// TIA Portal project "Vagoneta-1516" (V15.1)

(* hardware
DEVICE "S71500/ET200MP station_1"  S7-1500 station
   slot 0: "Perfil soporte_0"  Rack  6ES7 590-1***0-0AA0
   slot 1: "PLC_1"  CPU 1516-3 PN/DP  6ES7 516-3AN01-0AB0  V2.6
      slot 3: "Display de la CPU_1"  6ES7591-1BA00-0AA0
*)

// ===== PLC "PLC_1"  CPU 1516-3 PN/DP =====

VAR_GLOBAL   // PLC tag table "Tabla de variables estándar"
   "E0-Reposo" AT %M10.0 : Bool;
   "E1-avance_a_carga" AT %M10.1 : Bool;
   "E2-carga" AT %M10.2 : Bool;
   "E3-avance_a_descarga" AT %M10.3 : Bool;
   "E4-descarga" AT %M10.4 : Bool;
   "P_marcha" AT %I0.0 : Bool;
   "FC1_inicio" AT %I0.1 : Bool;
   "FC2_carga" AT %I0.2 : Bool;
   "FC3_descarga" AT %I0.3 : Bool;
   "Luz_verde" AT %Q0.0 : Bool;
   "Luz_roja" AT %Q0.1 : Bool;
   "Valvula" AT %Q0.2 : Bool;
   "E5-retroceso" AT %M10.5 : Bool;
   "Tag_1" AT %M50.0 : Bool;
   "Tag_2" AT %M50.1 : Bool;
   "Tag_3" AT %M50.2 : Bool;
   "P_Paro" AT %I0.4 : Bool;
   "Motor_avanza" AT %Q0.3 : Bool;
   "Motor_retrocede" AT %Q0.4 : Bool;
   "Zumbador" AT %Q0.5 : Bool;
   "Error_www" AT %MW100 : Int;
   "ContadorCiclos" AT %MB102 : SInt;
   "Tag_4" AT %M50.6 : Bool;
   "Tag_5" AT %M50.3 : Bool;
   "Estado" AT %MB103 : SInt;
   "Tag_6" AT %M70.0 : Bool;
   "Tag_7" AT %M70.1 : Bool;
   "Tag_8" AT %M70.2 : Bool;
   "Tag_9" AT %M70.3 : Bool;
   "Tag_10" AT %M70.4 : Bool;
   "Tag_11" AT %M70.5 : Bool;
   "System_Byte" AT %MB1 : Byte;
   "FirstScan" AT %M1.0 : Bool;
   "DiagStatusUpdate" AT %M1.1 : Bool;
   "AlwaysTRUE" AT %M1.2 : Bool;
   "AlwaysFALSE" AT %M1.3 : Bool;
   "tCarga" AT %MW104 : Int;
   "tDescarga" AT %MW106 : Int;
END_VAR

// folder: System blocks/Program resources

DATA_BLOCK "TP_5s"   // DB1
{ S7_Optimized_Access := 'TRUE' }
AUTHOR : Simatic
FAMILY : IEC
NAME : IEC_TMR
VERSION : 1.0
// stored: InstanceOfName IEC_TIMER
"IEC_TIMER"
BEGIN
END_DATA_BLOCK

DATA_BLOCK "TP_descarga"   // DB2
{ S7_Optimized_Access := 'TRUE' }
AUTHOR : Simatic
FAMILY : IEC
NAME : IEC_TMR
VERSION : 1.0
// stored: InstanceOfName IEC_TIMER
"IEC_TIMER"
BEGIN
END_DATA_BLOCK

DATA_BLOCK "CTU_ciclos"   // DB3
{ S7_Optimized_Access := 'TRUE' }
AUTHOR : Simatic
FAMILY : IEC
NAME : CNTR
VERSION : 1.0
// stored: InstanceOfName IEC_COUNTER
"IEC_COUNTER"
BEGIN
END_DATA_BLOCK

// folder: (top level)

ORGANIZATION_BLOCK "Main"   // OB1, LAD, ProgramCycle
TITLE = "Main Program Sweep (Cycle)"
{ S7_Optimized_Access := 'TRUE' }
VERSION : 0.1
   VAR_INPUT
      Initial_Call : Bool;   // Initial call of this OB
      Remanence : Bool;   // =True, if remanent data are available
   END_VAR
   VAR_TEMP   // added for the SCL form of the ladder/FBD networks
      _w1 : Bool;
      _w2 : Bool;
   END_VAR
BEGIN

REGION Network 1: Activar WWW
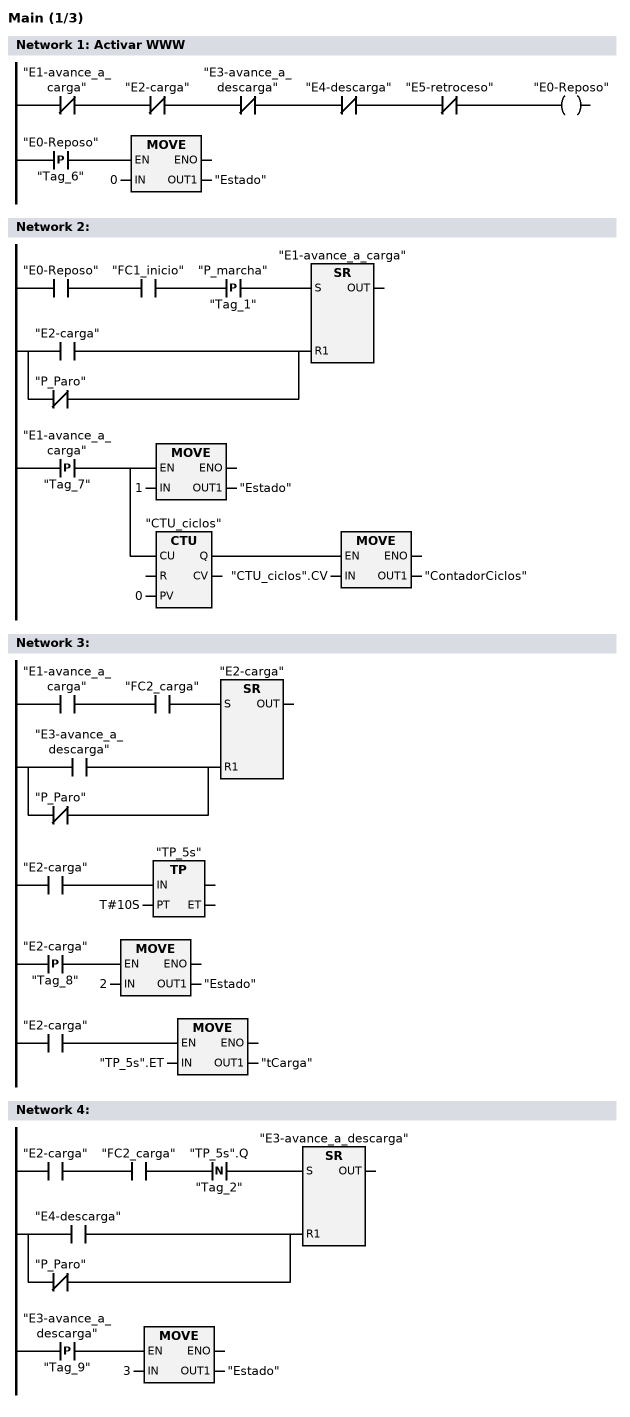
   RUNG wire#powerrail
      I_Contact( "E1-avance_a_carga" )
      I_Contact( "E2-carga" )
      I_Contact( "E3-avance_a_descarga" )
      I_Contact( "E4-descarga" )
      I_Contact( "E5-retroceso" )
      Coil( "E0-Reposo" )
   END_RUNG
   RUNG wire#powerrail
      P_Contact(operand := "E0-Reposo", bit := "Tag_6")
      Move(in := 0, out1 => "Estado")
   END_RUNG
   // the same network as SCL:
   "E0-Reposo" := NOT "E1-avance_a_carga" AND NOT "E2-carga" AND NOT "E3-avance_a_descarga" AND NOT "E4-descarga" AND NOT "E5-retroceso";
   #_w1 := "E0-Reposo" AND NOT "Tag_6";   // rising edge of "E0-Reposo"
   "Tag_6" := "E0-Reposo";
   IF #_w1 THEN "Estado" := 0; END_IF;
END_REGION

REGION Network 2
   #_w1 := "E0-Reposo" AND "FC1_inicio" AND "P_marcha" AND NOT "Tag_1";   // rising edge of "P_marcha"
   "Tag_1" := "P_marcha";
   IF #_w1 THEN
       "E1-avance_a_carga" := TRUE;   // SR flip-flop
   END_IF;
   IF "E2-carga" OR NOT "P_Paro" THEN "E1-avance_a_carga" := FALSE; END_IF;
   #_w2 := "E1-avance_a_carga" AND NOT "Tag_7";   // rising edge of "E1-avance_a_carga"
   "Tag_7" := "E1-avance_a_carga";
   IF #_w2 THEN "Estado" := 1; END_IF;
   "CTU_ciclos".CTU(CU := #_w2, PV := 0);
   IF "CTU_ciclos".Q THEN "ContadorCiclos" := "CTU_ciclos".CV; END_IF;
END_REGION

REGION Network 3
   IF "E1-avance_a_carga" AND "FC2_carga" THEN
       "E2-carga" := TRUE;   // SR flip-flop
   END_IF;
   IF "E3-avance_a_descarga" OR NOT "P_Paro" THEN "E2-carga" := FALSE; END_IF;
   "TP_5s".TP(IN := "E2-carga", PT := T#10S);
   #_w1 := "E2-carga" AND NOT "Tag_8";   // rising edge of "E2-carga"
   "Tag_8" := "E2-carga";
   IF #_w1 THEN "Estado" := 2; END_IF;
   IF "E2-carga" THEN "tCarga" := "TP_5s".ET; END_IF;
END_REGION

REGION Network 4
   RUNG wire#powerrail
      Contact( "E2-carga" )
      Contact( "FC2_carga" )
      N_Contact(operand := "TP_5s".Q, bit := "Tag_2")
      S_SR(operand := "E3-avance_a_descarga", r1 := wire#w1)
   END_RUNG
   RUNG wire#powerrail
      Contact( "E4-descarga" )
   END_RUNG wire#w1
   RUNG wire#powerrail
      I_Contact( "P_Paro" )
   END_RUNG wire#w1
   RUNG wire#powerrail
      P_Contact(operand := "E3-avance_a_descarga", bit := "Tag_9")
      Move(in := 3, out1 => "Estado")
   END_RUNG
   // the same network as SCL:
   #_w1 := "E2-carga" AND "FC2_carga" AND NOT "TP_5s".Q AND "Tag_2";   // falling edge of "TP_5s".Q
   "Tag_2" := "TP_5s".Q;
   IF #_w1 THEN
       "E3-avance_a_descarga" := TRUE;   // SR flip-flop
   END_IF;
   IF "E4-descarga" OR NOT "P_Paro" THEN "E3-avance_a_descarga" := FALSE; END_IF;
   #_w2 := "E3-avance_a_descarga" AND NOT "Tag_9";   // rising edge of "E3-avance_a_descarga"
   "Tag_9" := "E3-avance_a_descarga";
   IF #_w2 THEN "Estado" := 3; END_IF;
END_REGION

REGION Network 5
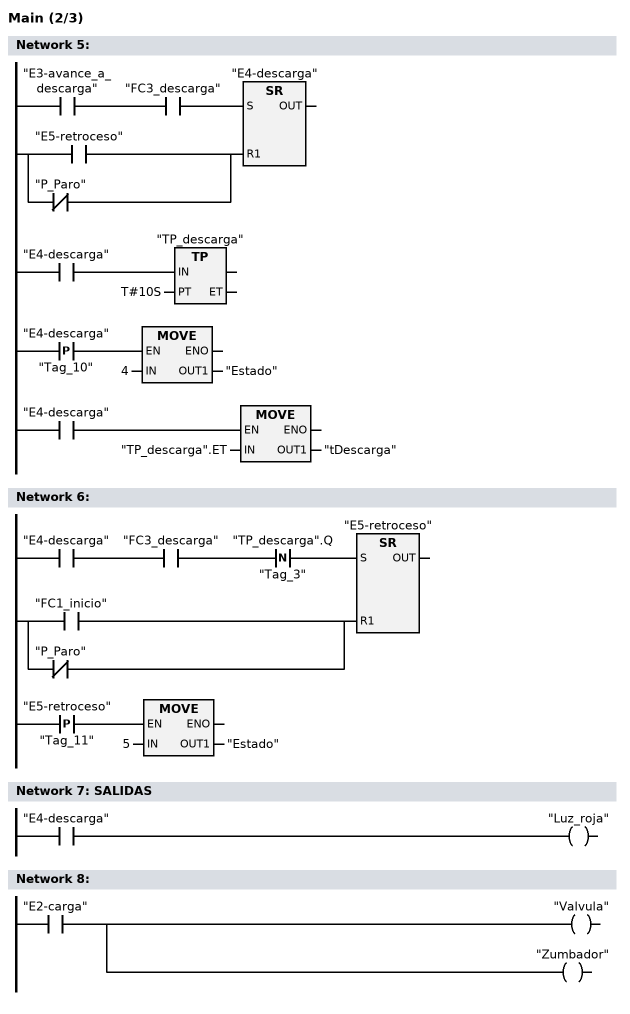
   IF "E3-avance_a_descarga" AND "FC3_descarga" THEN
       "E4-descarga" := TRUE;   // SR flip-flop
   END_IF;
   IF "E5-retroceso" OR NOT "P_Paro" THEN "E4-descarga" := FALSE; END_IF;
   "TP_descarga".TP(IN := "E4-descarga", PT := T#10S);
   #_w1 := "E4-descarga" AND NOT "Tag_10";   // rising edge of "E4-descarga"
   "Tag_10" := "E4-descarga";
   IF #_w1 THEN "Estado" := 4; END_IF;
   IF "E4-descarga" THEN "tDescarga" := "TP_descarga".ET; END_IF;
END_REGION

REGION Network 6
   RUNG wire#powerrail
      Contact( "E4-descarga" )
      Contact( "FC3_descarga" )
      N_Contact(operand := "TP_descarga".Q, bit := "Tag_3")
      S_SR(operand := "E5-retroceso", r1 := wire#w1)
   END_RUNG
   RUNG wire#powerrail
      Contact( "FC1_inicio" )
   END_RUNG wire#w1
   RUNG wire#powerrail
      I_Contact( "P_Paro" )
   END_RUNG wire#w1
   RUNG wire#powerrail
      P_Contact(operand := "E5-retroceso", bit := "Tag_11")
      Move(in := 5, out1 => "Estado")
   END_RUNG
   // the same network as SCL:
   #_w1 := "E4-descarga" AND "FC3_descarga" AND NOT "TP_descarga".Q AND "Tag_3";   // falling edge of "TP_descarga".Q
   "Tag_3" := "TP_descarga".Q;
   IF #_w1 THEN
       "E5-retroceso" := TRUE;   // SR flip-flop
   END_IF;
   IF "FC1_inicio" OR NOT "P_Paro" THEN "E5-retroceso" := FALSE; END_IF;
   #_w2 := "E5-retroceso" AND NOT "Tag_11";   // rising edge of "E5-retroceso"
   "Tag_11" := "E5-retroceso";
   IF #_w2 THEN "Estado" := 5; END_IF;
END_REGION

REGION Network 7: SALIDAS
   RUNG wire#powerrail
      Contact( "E4-descarga" )
      Coil( "Luz_roja" )
   END_RUNG
   // the same network as SCL:
   "Luz_roja" := "E4-descarga";
END_REGION

REGION Network 8
   RUNG wire#powerrail
      Contact( "E2-carga" )
      wire#w1
      Coil( "Valvula" )
   END_RUNG
   RUNG wire#w1
      Coil( "Zumbador" )
   END_RUNG
   // the same network as SCL:
   "Valvula" := "E2-carga";
   "Zumbador" := "E2-carga";
END_REGION

REGION Network 9
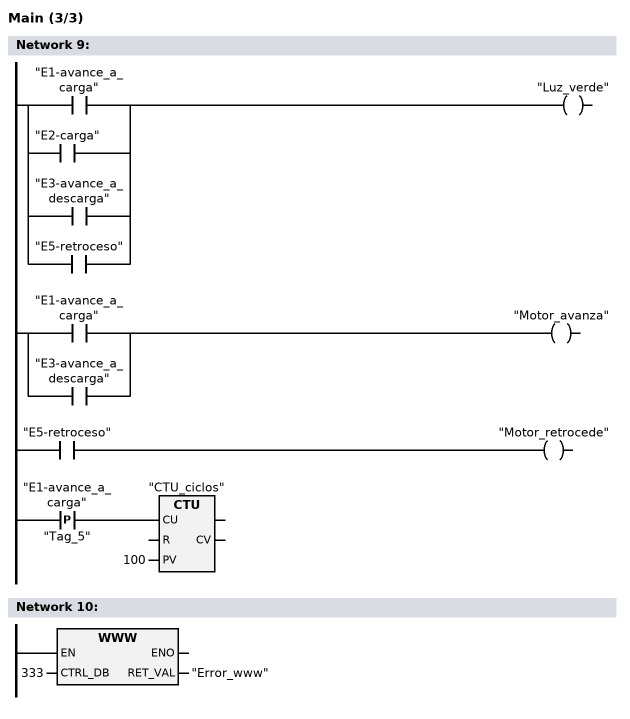
   "Luz_verde" := "E1-avance_a_carga" OR "E2-carga" OR "E3-avance_a_descarga" OR "E5-retroceso";
   "Motor_avanza" := "E1-avance_a_carga" OR "E3-avance_a_descarga";
   "Motor_retrocede" := "E5-retroceso";
   #_w1 := "E1-avance_a_carga" AND NOT "Tag_5";   // rising edge of "E1-avance_a_carga"
   "Tag_5" := "E1-avance_a_carga";
   "CTU_ciclos".CTU(CU := #_w1, PV := 100);
END_REGION

REGION Network 10
   "Error_www" := WWW(CTRL_DB := 333);
END_REGION
END_ORGANIZATION_BLOCK